# EPICS substitutions: evrSupport/Db/ioc/bsaAMPLEdef.substitutions
#==============================================================================
#
# Abs:  Beam Synchronous Acquisition records for a single
#	    RF Amplitude measurement.
#
# Name: bsaAMPLEdef.substitutions
#
# Note: Must follow the LCLS naming conventions.
#
#==============================================================================
#
#
file bsaATTREdef.db
{
#           Device   Attribute  Input  EGU   HOPR  LOPR PREC ADEL  Link
  pattern {   D       , ATTR   , I   , EG ,  HO  , LO , PR , AD  ,  LNK,      SINK_SIZE  }
	  { $(DEVICE) ,$(ATRB) ,$(IN), meV ,  0  ,  0 ,  3 , .01 , $(SLCLNK), $(SINK_SIZE\=10) }
}
